FUNCTION_BLOCK ReservoirTankDrainNIL
VAR_INPUT

	bMainOnOff:BOOL;
	iDrainCollectTimer:INT;
	iDrainTransferTimer:INT;
	iDrainingTimer:INT;
	bDirectDrainST:BOOL;
END_VAR

VAR_OUTPUT

	bReservoirDrainAv1:BOOL;
	bReservoirDrainAv2:BOOL;
	ProcessComplete:BOOL;
END_VAR

VAR
	Timer1: DOWN_COUNT_TIMER;
	CollectTimerComplete: BOOL;
	Timer2: DOWN_COUNT_TIMER;
	TransferComplete: BOOL;
	Timer3: DOWN_COUNT_TIMER;
	DrainComplete: BOOL;
	DelayComplete: TON;
	Coundown: INT;
	bDirectDrainInProcess: BOOL;
END_VAR

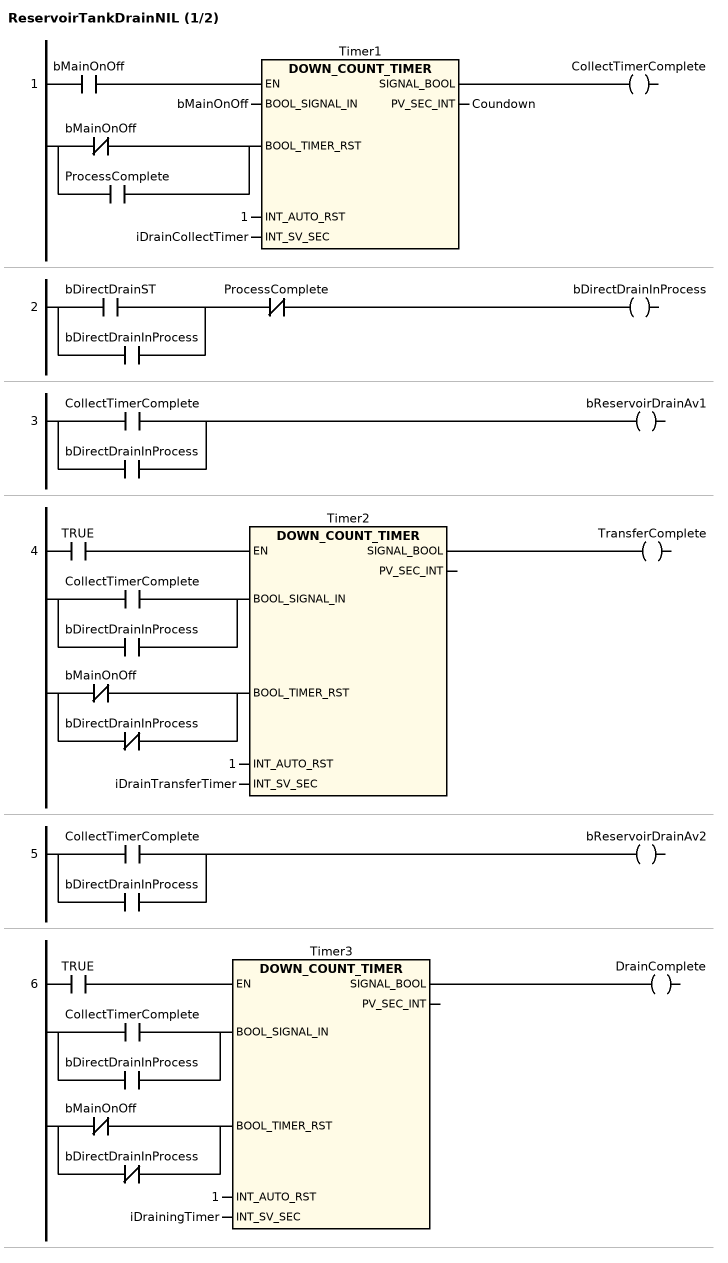
// NETWORK 1
IF bMainOnOff THEN
    Timer1(
        BOOL_SIGNAL_IN := bMainOnOff,
        BOOL_TIMER_RST := NOT bMainOnOff OR ProcessComplete,
        INT_AUTO_RST := 1,
        INT_SV_SEC := iDrainCollectTimer,
        PV_SEC_INT => Coundown); // DOWN_COUNT_TIMER
END_IF
CollectTimerComplete := Timer1.SIGNAL_BOOL;

// NETWORK 2
bDirectDrainInProcess := (bDirectDrainST OR bDirectDrainInProcess) AND NOT ProcessComplete;

// NETWORK 3
bReservoirDrainAv1 := CollectTimerComplete OR bDirectDrainInProcess;

// NETWORK 4
Timer2(
    BOOL_SIGNAL_IN := CollectTimerComplete OR bDirectDrainInProcess,
    BOOL_TIMER_RST := NOT bMainOnOff OR NOT bDirectDrainInProcess,
    INT_AUTO_RST := 1,
    INT_SV_SEC := iDrainTransferTimer); // DOWN_COUNT_TIMER
TransferComplete := Timer2.SIGNAL_BOOL;

// NETWORK 5
bReservoirDrainAv2 := CollectTimerComplete OR bDirectDrainInProcess;

// NETWORK 6
Timer3(
    BOOL_SIGNAL_IN := CollectTimerComplete OR bDirectDrainInProcess,
    BOOL_TIMER_RST := NOT bMainOnOff OR NOT bDirectDrainInProcess,
    INT_AUTO_RST := 1,
    INT_SV_SEC := iDrainingTimer); // DOWN_COUNT_TIMER
DrainComplete := Timer3.SIGNAL_BOOL;

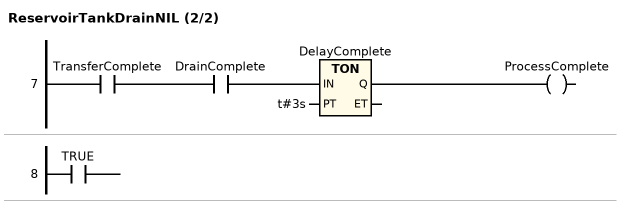
// NETWORK 7
DelayComplete(IN := TransferComplete AND DrainComplete, PT := t#3s); // TON
ProcessComplete := DelayComplete.Q;

// NETWORK 8

END_FUNCTION_BLOCK

(* stored: Version 1.1.0.1, ProductVersion 3.1.4024.12
   POU ReservoirTankDrainNIL: Id {b0b93ca5-f910-42bd-a5dd-46707123cea0}, SpecialFunc None *)
